RoboDK station: RecoverPrograms.rdk

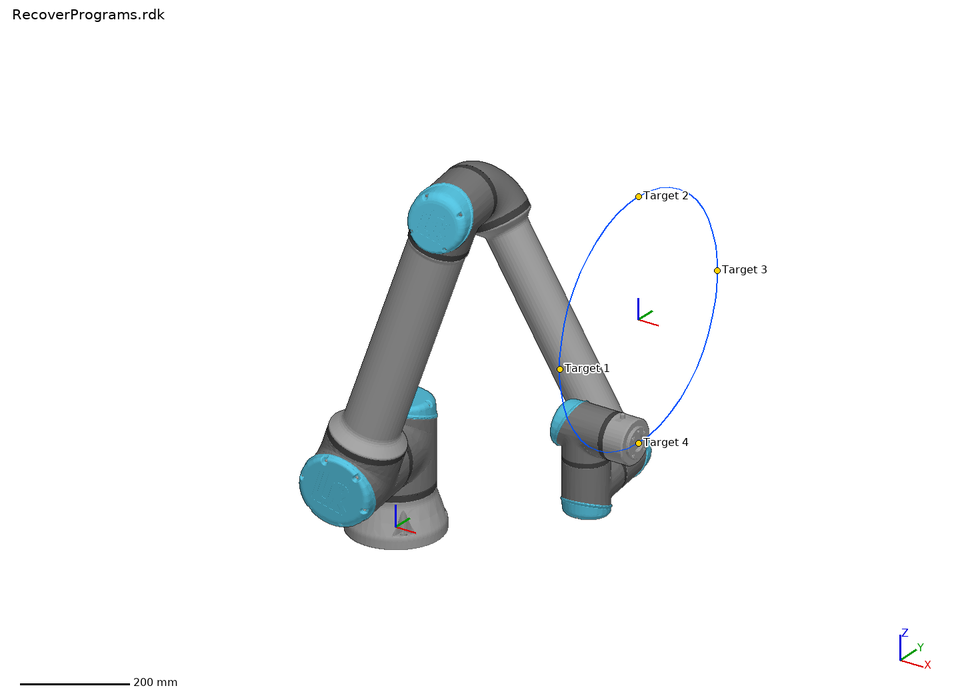
[picture v0: the station drawn from its stored meshes, robots at their saved joint values, targets as dots, program paths as lines]
Station RecoverPrograms (saved by RoboDK 5.5.2). Poses are relative to the parent item; angles as X-Y-Z fixed-axis rotations.
Station parameters (name, value as stored): ProgUtilities-Settings
  - frame UR10e Base at (0, 0, 0) mm
    - robot UR10e: 6 axes, payload 10 kg, reach 1300 mm, repeatability 0.05 mm, weight 28.9 kg
        modified DH rows (alpha deg, a mm, theta deg, d mm): 0, 0, 0, 180.7; 90, 0, 180, 0; 0, 612.6, 0, 0; 0, 571.335, 0, 174.15; -90, 0, 0, 119.85; 90, 0, 180, 116.55
        joint limits [-360, -360, -360, -360, -360, -360] to [360, 360, 360, 360, 360, 360]; home [0, -90, -90, 0, 90, 0]; saved at [8.78, -108.762, -132.424, 61.186, 81.22, 0]
    - frame Frame 2 at (610, -100, 630) mm
      - target Target 1 (Cartesian target) at (0, -250, 0) mm, rotated rx -90 ry 0 rz -90 deg; joints [-18.618, -97.519, -111.584, 29.103, 108.618, 0] of UR10e
      - target Target 2 (Cartesian target) at (0, 0, 250) mm, rotated rx -90 ry 0 rz -90 deg; joints [8.78, -80.759, -101.769, 2.528, 81.22, 0] of UR10e
      - target Target 3 (Cartesian target) at (0, 250, 0) mm, rotated rx -90 ry 0 rz -90 deg; joints [36.643, -88.986, -120.711, 29.698, 53.357, 0] of UR10e
      - target Target 4 (Cartesian target) at (0, 0, -250) mm, rotated rx -90 ry 0 rz -90 deg; joints [8.78, -108.762, -132.424, 61.186, 81.22, 0] of UR10e
  - program Prog1 (4 instructions, listed below)
  - program Prog1 Recovered (4 instructions, listed below)

--- program Prog1 ---
  Set Ref.: Frame 2 at (610, -100, 630) mm
  MoveJ (Target 4) [its target is no longer in the station]
  MoveC (Target 1, Target 2) [its target is no longer in the station] [its target is no longer in the station]
  MoveC (Target 3, Target 4) [its target is no longer in the station] [its target is no longer in the station]

--- program Prog1 Recovered (robot UR10e) ---
  Set Ref.: Frame 2
  MoveJ (Target 4)
  MoveC (Target 1, Target 2)
  MoveC (Target 3, Target 4)
